Universal Robots PolyScope program: sandFront.urp

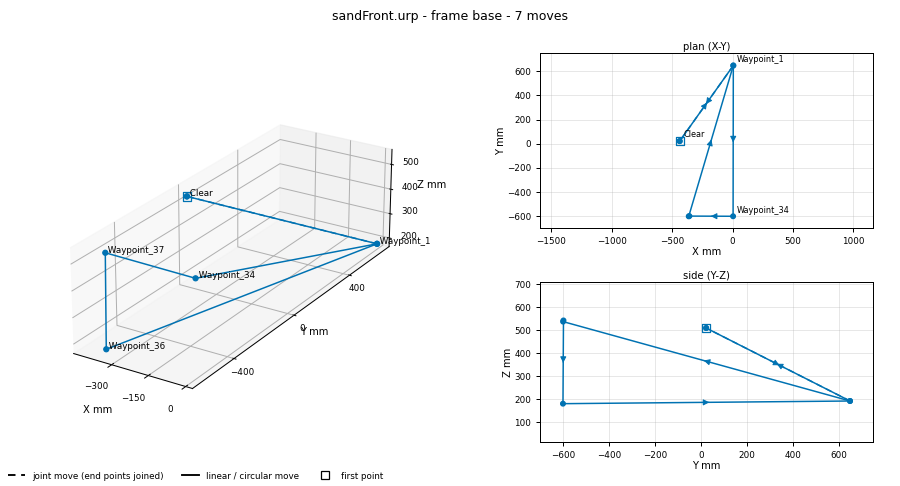
[picture p0: tool path of sandFront.urp in frame base, 7 of 7 moves have a stored position in this frame; points joined in program order, loops and branches not executed]
Program sandFront (installation=sand5 directory=/programs/subs createdIn=5.11.5.1010327 lastSavedIn=5.11.5.1010327 robotSerialNumber=20215500677)
Calibrated DH parameters: a=[0.000204, -0.239222, -0.391845, -0.000001, 0.000022, 0]; d=[0.162722, -355.808559, 353.37206, 2.570385, 0.099741, 0.099629]; alpha=[1.571124, 0.000988, 0.008295, 1.568963, -1.570303, 0]; deltaTheta=[0, -0.973091, 7.204745, 0.05153, 0, 0]
Robot Program (runOnlyOnce=false)
  Folder sandFront
    MoveJ speed 60 deg/s, acceleration 80 deg/s^2 (useActiveTCP=false positionType=JointAngles) tcp=DynabradeDual; feature=Work
      Waypoint Clear: TCP in base x=-437.78 y=22.317 z=510.388 mm, rx=-1.2261 ry=-1.1914 rz=1.1915 rad; joints [-41.645, -103.017, 131.059, 99.527, -63.29, 31.09] deg; TCP offset x=3.18 y=114.64 z=98.2 mm, rx=-0.7854 ry=0 rz=0 rad; feature pose in base x=-591.611 y=-180.941 z=285.211 mm, rx=1.216 ry=1.1897 rz=1.1897 rad
      SuppressedNode
        Waypoint Waypoint_35: TCP in base x=-544.551 y=45.618 z=509.072 mm, rx=-1.2092 ry=-1.2181 rz=1.2109 rad; joints [-31.988, -85.182, 115.602, 99.979, -68.031, 24.222] deg; TCP offset x=3.18 y=114.64 z=98.2 mm, rx=-0.7854 ry=0 rz=0 rad; feature pose in base x=-691.483 y=-161.421 z=282.725 mm, rx=1.203 ry=1.2097 rz=1.2171 rad
    MoveL speed 250 mm/s, acceleration 1200 mm/s^2 (useActiveTCP=false) tcp=DynabradeDual; feature=Work
      Waypoint Waypoint_1: TCP in base x=6.072 y=648.1 z=192.982 mm, rx=-1.5699 ry=0.0092 rz=0.0097 rad; joints [251.403, -67.593, 131.535, -110.394, 77.851, -166.352] deg; feature pose in base x=6.058 y=653.089 z=192.929 mm, rx=1.5716 ry=0.003 rz=-0.0025 rad
      URCap Zero FT Sensor (Robotiq_Copilot, Robotiq Inc.) dataModel(NodeInitializedKey=true, WaitForSteadyWrenchOptionKey=true)
      URCap Find Surface (Robotiq_Copilot, Robotiq Inc.) dataModel(NodeInitializedKey=true, WaitForSteadyWrenchOptionKey=false, ls_force=10.0, ls_distance=100.0, ls_speed=5.0, ZeroSensorBeforeKey=false, ls_if_distance=false, ls_if_force=false); state(isChildrenLocked=true)
        'Add Stop conditions from the Find Surface node'
      URCap Finishing Tool Control (Robotiq_Copilot, Robotiq Inc.) dataModel(ToolOutputNameKey=digital_out[0], HackTriggeringContributionIsDefinedMethodKey=true)
      Wait Sleep waitTime=0.5
    MoveL speed 60 mm/s, acceleration 1200 mm/s^2 (useActiveTCP=false) tcp=DynabradeDual; feature=Work
      Force Simple feature=Joint_6_name; selection=[0, 0, 1, 0, 0, 0]; wrench=[0, 0, 7, 0, 0, 0]; limitsForce=[0.15, 0.15, 0.15, 1.047198, 1.047198, 1.047198]; limitsMotion=[0.1, 0.1, 0.1, 0.349066, 0.349066, 0.349066]
        Waypoint Waypoint_34: TCP in base x=4.168 y=-599.662 z=538.228 mm, rx=0.1003 ry=-2.1628 rz=2.1762 rad; joints [69.8, -105.08, 109.114, -52.157, 72.617, -168.988] deg; feature pose in base x=2.048 y=-607.004 z=173.227 mm, rx=-0.0204 ry=-2.2235 rz=-2.2094 rad
        Waypoint Waypoint_37: TCP in base x=-357.721 y=-598.101 z=543.274 mm, rx=0.1002 ry=-2.1629 rz=2.1762 rad; joints [31.577, -86.57, 95.791, -75.508, 51.138, -132.637] deg
        Waypoint Waypoint_36: TCP in base x=-362.939 y=-600.337 z=181.342 mm, rx=0.1002 ry=-2.1628 rz=2.1761 rad; joints [31.404, -55.313, 118.507, -129.285, 51.013, -132.956] deg
        Waypoint Waypoint_1: TCP in base x=6.072 y=648.1 z=192.982 mm, rx=-1.5699 ry=0.0092 rz=0.0097 rad; joints [251.403, -67.593, 131.535, -110.394, 77.851, -166.352] deg; feature pose in base x=6.058 y=653.089 z=192.929 mm, rx=1.5716 ry=0.003 rz=-0.0025 rad
        URCap Finishing Tool Control (Robotiq_Copilot, Robotiq Inc.) dataModel(FinishingToolStateKey=false, ToolOutputNameKey=digital_out[0], HackTriggeringContributionIsDefinedMethodKey=true)
      MoveDirectionNode (selectedDirection=ZMinus) feature=Joint_6_name
        Until DISTANCE (allowActions=false deceleration=3 distanceNodeType=STOP) Distance=0.025; motionParameters(blendRadius=0)
    MoveJ speed 60 deg/s, acceleration 80 deg/s^2 (useActiveTCP=true positionType=JointAngles) feature=Work
      Waypoint Clear: TCP in base x=-437.78 y=22.317 z=510.388 mm, rx=-1.2261 ry=-1.1914 rz=1.1915 rad; joints [-41.645, -103.017, 131.059, 99.527, -63.29, 31.09] deg; TCP offset x=3.18 y=114.64 z=98.2 mm, rx=-0.7854 ry=0 rz=0 rad; feature pose in base x=-591.611 y=-180.941 z=285.211 mm, rx=1.216 ry=1.1897 rz=1.1897 rad
      SuppressedNode
        Waypoint Waypoint_35: TCP in base x=-544.551 y=45.618 z=509.072 mm, rx=-1.2092 ry=-1.2181 rz=1.2109 rad; joints [-31.988, -85.182, 115.602, 99.979, -68.031, 24.222] deg; TCP offset x=3.18 y=114.64 z=98.2 mm, rx=-0.7854 ry=0 rz=0 rad; feature pose in base x=-691.483 y=-161.421 z=282.725 mm, rx=1.203 ry=1.2097 rz=1.2171 rad
